TYPE SampleArrayToRender :
STRUCT
	Data	:	ARRAY  [0..100] OF SampleDataItem;
END_STRUCT
END_TYPE

(* stored: Version 1.1.0.1
   DUT SampleArrayToRender: Id {0fdee56a-6183-4123-afd7-208a33986db7} *)
